(* CODESYS project MPS2017.project

Project tree, tasks and I/O mapping:
  Device : CECC-LK, Festo AG & Co. KG, order no. 574418, version 3.5.7.27
    application Application
      task Task (cyclic, interval 100 ms, priority 20) calls POU
      program POU [ST]
      global variables GVL
    Onboard : CECC 14I/8O, Festo AG & Co. KG, version 3.4.5.5
        unmapped channels: Onboard Input, Onboard Output
      Digital Inputs
          unmapped channels: Onboard Input
      Digital Outputs
          unmapped channels: Onboard Output
    Ethernet : Ethernet, 3S - Smart Software Solutions GmbH, version 3.5.7.0
        settings: IPAddress = [192,168,2,28]; SubnetMask = [255,255,255,0]; GatewayAddress = [0,0,0,0]; MACAddress = [16#00,16#00,16#00,16#00,16#00,16#00]; NetworkInterfaceName = 'eth0'; NetworkInterfaceName = "eth0"
      ModbusTCP_Slave_Device : ModbusTCP Slave Device, 3S - Smart Software Solutions GmbH, version 3.5.10.0
          settings: Unit-ID = 1; Data Model Options = 1
          input  Application.input1 AT %IW10 : ARRAY[0..11] OF WORD  // Inputs
          output Application.output1 AT %QW10 : ARRAY[0..11] OF WORD  // Outputs
    IO_Link_Master_4_Ports_ : IO-Link Master (4 Ports), Festo AG & Co. KG, order no. 
      , version 3.0.0.3
      BNI_IOL_310_000_K025 : BNI IOL-310-000-K025, BALLUFF, version V1.3
          settings:  = 0; ProcessDataID = V_PdT; ProcessDataInLength = 16; ProcessDataOutLength = 16; ProcessDataDescription.bitOffset = 8; ProcessDataDescription.bitLength = 1; ProcessDataDescription.userType = 0; ProcessDataDescription.ChannelType = 1; ProcessDataDescription.TotalLength = 16; ProcessDataDescription.bitOffset = 9; ProcessDataDescription.bitLength = 1; ProcessDataDescription.userType = 0; ProcessDataDescription.ChannelType = 1; ProcessDataDescription.TotalLength = 16; ProcessDataDescription.bitOffset = 10; ProcessDataDescription.bitLength = 1; ProcessDataDescription.userType = 0; ProcessDataDescription.ChannelType = 1; ProcessDataDescription.TotalLength = 16; ProcessDataDescription.bitOffset = 11; ProcessDataDescription.bitLength = 1; ProcessDataDescription.userType = 0; ProcessDataDescription.ChannelType = 1; ProcessDataDescription.TotalLength = 16; ProcessDataDescription.bitOffset = 12; ProcessDataDescription.bitLength = 1; ProcessDataDescription.userType = 0; ProcessDataDescription.ChannelType = 1; ProcessDataDescription.TotalLength = 16; ProcessDataDescription.bitOffset = 13; ProcessDataDescription.bitLength = 1; ProcessDataDescription.userType = 0; ProcessDataDescription.ChannelType = 1; ProcessDataDescription.TotalLength = 16; ProcessDataDescription.bitOffset = 14; ProcessDataDescription.bitLength = 1; ProcessDataDescription.userType = 0; ProcessDataDescription.ChannelType = 1; ProcessDataDescription.TotalLength = 16; ProcessDataDescription.bitOffset = 15;
            ProcessDataDescription.bitLength = 1; ProcessDataDescription.userType = 0; ProcessDataDescription.ChannelType = 1; ProcessDataDescription.TotalLength = 16; ProcessDataDescription.bitOffset = 0; ProcessDataDescription.bitLength = 1; ProcessDataDescription.userType = 0; ProcessDataDescription.ChannelType = 1; ProcessDataDescription.TotalLength = 16; ProcessDataDescription.bitOffset = 1; ProcessDataDescription.bitLength = 1; ProcessDataDescription.userType = 0; ProcessDataDescription.ChannelType = 1; ProcessDataDescription.TotalLength = 16; ProcessDataDescription.bitOffset = 2; ProcessDataDescription.bitLength = 1; ProcessDataDescription.userType = 0; ProcessDataDescription.ChannelType = 1; ProcessDataDescription.TotalLength = 16; ProcessDataDescription.bitOffset = 3; ProcessDataDescription.bitLength = 1; ProcessDataDescription.userType = 0; ProcessDataDescription.ChannelType = 1; ProcessDataDescription.TotalLength = 16; ProcessDataDescription.bitOffset = 4; ProcessDataDescription.bitLength = 1; ProcessDataDescription.userType = 0; ProcessDataDescription.ChannelType = 1; ProcessDataDescription.TotalLength = 16; ProcessDataDescription.bitOffset = 5; ProcessDataDescription.bitLength = 1; ProcessDataDescription.userType = 0; ProcessDataDescription.ChannelType = 1; ProcessDataDescription.TotalLength = 16; ProcessDataDescription.bitOffset = 6; ProcessDataDescription.bitLength = 1; ProcessDataDescription.userType = 0; ProcessDataDescription.ChannelType = 1; ProcessDataDescription.TotalLength = 16; ProcessDataDescription.bitOffset = 7;
            ProcessDataDescription.bitLength = 1; ProcessDataDescription.userType = 0; ProcessDataDescription.ChannelType = 1; ProcessDataDescription.TotalLength = 16; ProcessDataDescription.bitOffset = 8; ProcessDataDescription.bitLength = 1; ProcessDataDescription.userType = 0; ProcessDataDescription.ChannelType = 2; ProcessDataDescription.TotalLength = 16; ProcessDataDescription.bitOffset = 9; ProcessDataDescription.bitLength = 1; ProcessDataDescription.userType = 0; ProcessDataDescription.ChannelType = 2; ProcessDataDescription.TotalLength = 16; ProcessDataDescription.bitOffset = 10; ProcessDataDescription.bitLength = 1; ProcessDataDescription.userType = 0; ProcessDataDescription.ChannelType = 2; ProcessDataDescription.TotalLength = 16; ProcessDataDescription.bitOffset = 11; ProcessDataDescription.bitLength = 1; ProcessDataDescription.userType = 0; ProcessDataDescription.ChannelType = 2; ProcessDataDescription.TotalLength = 16; ProcessDataDescription.bitOffset = 12; ProcessDataDescription.bitLength = 1; ProcessDataDescription.userType = 0; ProcessDataDescription.ChannelType = 2; ProcessDataDescription.TotalLength = 16; ProcessDataDescription.bitOffset = 13; ProcessDataDescription.bitLength = 1; ProcessDataDescription.userType = 0; ProcessDataDescription.ChannelType = 2; ProcessDataDescription.TotalLength = 16; ProcessDataDescription.bitOffset = 14; ProcessDataDescription.bitLength = 1; ProcessDataDescription.userType = 0; ProcessDataDescription.ChannelType = 2; ProcessDataDescription.TotalLength = 16; ProcessDataDescription.bitOffset = 15;
            ProcessDataDescription.bitLength = 1; ProcessDataDescription.userType = 0; ProcessDataDescription.ChannelType = 2; ProcessDataDescription.TotalLength = 16; ProcessDataDescription.bitOffset = 0; ProcessDataDescription.bitLength = 1; ProcessDataDescription.userType = 0; ProcessDataDescription.ChannelType = 2; ProcessDataDescription.TotalLength = 16; ProcessDataDescription.bitOffset = 1; ProcessDataDescription.bitLength = 1; ProcessDataDescription.userType = 0; ProcessDataDescription.ChannelType = 2; ProcessDataDescription.TotalLength = 16; ProcessDataDescription.bitOffset = 2; ProcessDataDescription.bitLength = 1; ProcessDataDescription.userType = 0; ProcessDataDescription.ChannelType = 2; ProcessDataDescription.TotalLength = 16; ProcessDataDescription.bitOffset = 3; ProcessDataDescription.bitLength = 1; ProcessDataDescription.userType = 0; ProcessDataDescription.ChannelType = 2; ProcessDataDescription.TotalLength = 16; ProcessDataDescription.bitOffset = 4; ProcessDataDescription.bitLength = 1; ProcessDataDescription.userType = 0; ProcessDataDescription.ChannelType = 2; ProcessDataDescription.TotalLength = 16; ProcessDataDescription.bitOffset = 5; ProcessDataDescription.bitLength = 1; ProcessDataDescription.userType = 0; ProcessDataDescription.ChannelType = 2; ProcessDataDescription.TotalLength = 16; ProcessDataDescription.bitOffset = 6; ProcessDataDescription.bitLength = 1; ProcessDataDescription.userType = 0; ProcessDataDescription.ChannelType = 2; ProcessDataDescription.TotalLength = 16; ProcessDataDescription.bitOffset = 7;
            ProcessDataDescription.bitLength = 1; ProcessDataDescription.userType = 0; ProcessDataDescription.ChannelType = 2; ProcessDataDescription.TotalLength = 16
          unmapped channels: Switchstate Pin 1 (Bit0.0), Switchstate Pin 2 (Bit0.1), Switchstate Pin 3 (Bit0.2), Switchstate Pin 4 (Bit0.3), Switchstate Pin 5 (Bit0.4), Switchstate Pin 6 (Bit0.5), Switchstate Pin 7 (Bit0.6), Switchstate Pin 8 (Bit0.7), Switchstate Pin 9 (Bit1.0), Switchstate Pin 10 (Bit1.1), Switchstate Pin 11 (Bit1.2), Switchstate Pin 12 (Bit1.3), Switchstate Pin 13 (Bit1.4), Switchstate Pin 14 (Bit1.5), Switchstate Pin 15 (Bit1.6), Switchstate Pin 16 (Bit1.7), Switchstate Pin 1 (Bit0.0), Switchstate Pin 2 (Bit0.1), Switchstate Pin 3 (Bit0.2), Switchstate Pin 4 (Bit0.3), Switchstate Pin 5 (Bit0.4), Switchstate Pin 6 (Bit0.5), Switchstate Pin 7 (Bit0.6), Switchstate Pin 8 (Bit0.7), Switchstate Pin 9 (Bit1.0), Switchstate Pin 10 (Bit1.1), Switchstate Pin 11 (Bit1.2), Switchstate Pin 12 (Bit1.3), Switchstate Pin 13 (Bit1.4), Switchstate Pin 14 (Bit1.5), Switchstate Pin 15 (Bit1.6), Switchstate Pin 16 (Bit1.7)
      <Empty>
      <Empty>
      <Empty>
*)

// Device/Application/GVL
(* 
	Author: Alain Rohr (hftm.ch) / (Original by David Masternak(Festo)) 
	Date: 28.01.2017
*)

VAR_GLOBAL
	(** Variable for base station **)
	
	(* Input variables *)
	bs_partAtIn         AT %IX0.4 : BOOL;  (* Is part available on the left/in side *)
	bs_partAtOut        AT %IX0.6 : BOOL;  (* Is part available on the right/out side *)
	bs_base1Av          AT %IX2.2 : BOOL;  (* Are workpieces at output1 available *)
	bs_base2Av          AT %IX2.6 : BOOL;  (* Are workpieces at output2 available *)
	bs_base3Av          AT %IX0.2 : BOOL;  (* Are workpieces at output3 available *)
	bs_b1Retracted      AT %IX2.0 : BOOL;  (* Is Base1 Slide retracted *)
	bs_b1Extracted      AT %IX2.1 : BOOL;  (* Is Base1 Slide retracted *)
	
	bs_b2Retracted      AT %IX2.4 : BOOL;  (* Is Base2 Slide retracted *)
	bs_b2Extracted      AT %IX2.5 : BOOL;  (* Is Base2 Slide retracted *)
	
	bs_b3Retracted      AT %IX0.0 : BOOL;  (* Is Base3 Slide retracted *)
	bs_b3Extracted      AT %IX0.1 : BOOL;  (* Is Base3 Slide retracted *)
	
	(* Output variables *)
	bs_output1          AT %QX2.0 : BOOL;  (* Get workpiece at output1 *)
	bs_output2          AT %QX2.4 : BOOL;  (* Get workpiece at output2 *)
	bs_output3          AT %QX0.0 : BOOL;  (* Get workpiece at output3 *)
	
	bs_motorToOut       AT %QX0.4 : BOOL;  (* Run bandmotor to the left side *)
	bs_motorToIn        AT %QX0.5 : BOOL;  (* Run bandmotor to the right side *)
	bs_lightRed         AT %QX2.5 : BOOL;  (* Red light *)
	bs_lightYellow      AT %QX2.6 : BOOL;  (* Yellow light *)
	bs_lightGreen       AT %QX2.7 : BOOL;  (* Green light *)

	(** Variable for Ring-Station (pick and place 2) **)

	(* Input variables *)
	rs_partAtIn         AT %IX2.0 : BOOL;  (* Part available *)
	rs_partAtSep        AT %IX2.1 : BOOL;  (* Part at seperator *)
	rs_partAtOut        AT %IX2.2 : BOOL;  (* Part at delivery *)
	rs_partAtSlide      AT %IX2.3 : BOOL;  (* Part at slide *)

	rs_slide1Retracted  AT %IX2.4 : BOOL;  (* is slide1 extracted *)
	rs_slide1Extracted  AT %IX2.5 : BOOL;  (* is slide2 extracted *)
    rs_vacuum1IsOn      AT %IX2.6 : BOOL;  (* Eco trigger for slide 1 *)    

    rs_slide2Retracted  AT %IX0.0 : BOOL;  (* is slide2 retracted *)	
    rs_slide2Extracted  AT %IX0.1 : BOOL;  (* is slide2 extracted *)	
	rs_vacuum2IsOn      AT %IX0.2 : BOOL;  (* Eco trigger for slide 2 *)
	
	(* Output variables *)
	rs_motorToOut       AT %QX2.0 : BOOL;  (* Turn on bandmotor to Out *)
	rs_seperator        AT %QX2.2 : BOOL;  (* Turn on seperator *)
	
	rs_slide1Retract    AT %QX2.4 : BOOL;  (* Retract slide 1 *)
	rs_slide1Extract    AT %QX2.5 : BOOL;  (* Extend slide 1 *)
	rs_slide1Down       AT %QX2.6 : BOOL;  (* Up/Down slide 1 *)
	rs_vacuum1On        AT %QX0.6 : BOOL;  (* Vacuum on at slide 1 *)
	rs_vacuum1Off       AT %QX0.7 : BOOL;  (* Vacuum off at slide 1 *)
	
	rs_slide2Retract    AT %QX0.0 : BOOL;  (* Retract slide 2 *)
	rs_slide2Extract    AT %QX0.1 : BOOL;  (* Extend slide 2 *)
	rs_slide2Down       AT %QX0.2 : BOOL;  (* Up/Down slide 2 *)
	rs_vacuum2On        AT %QX0.4 : BOOL;  (* Vacuum on at slide 2 *)
	rs_vacuum2Off       AT %QX0.5 : BOOL;  (* Vacuum off at slide 2 *)
	
	rs_lightRed         AT %QX0.3 : BOOL;  (* Red light *)
	rs_lightYellow      AT %QX2.6 : BOOL;  (* Yellow light *)
	rs_lightGreen       AT %QX2.7 : BOOL;  (* Green light *)
	

	(** Variable for Cap Station (pick and place 1) **)
	(* Input variables *)
    cs_vacuumIsOn       AT %IX0.0 : BOOL;  (* Is Eco trigger active *)	
    cs_partAtIn         AT %IX2.0 : BOOL;  (* Is part available *)
	cs_partAtSep        AT %IX2.1 : BOOL;  (* Is part at seperator *)
	cs_partAtOut	    AT %IX2.2 : BOOL;  (* Is part on delivery position *)
	cs_slideRetracted   AT %IX2.4 : BOOL;
	cs_slideExtracted   AT %IX2.5 : BOOL;
	cs_slideIsUp	    AT %IX2.6 : BOOL;  (*Cylinder Z-Achse*)
	
	(* Output variables *)
	cs_vacuumOn	        AT %QX0.0 : BOOL;  (* Turn on vacuum *)
	cs_vacuumOff        AT %QX0.1 : BOOL;  (* Turn off vacuum *)
	cs_lightRed         AT %QX0.5 : BOOL;  (* Red light *)
	cs_lightYellow      AT %QX0.6 : BOOL;  (* Yellow light *)
	cs_lightGreen       AT %QX0.7 : BOOL;  (* Green light *)
	
	cs_motorToOut       AT %QX2.0 : BOOL;  (* Bandmotor *)
	cs_motorToIn        AT %QX2.1 : BOOL;  (* Bandmotor in other direction *)
	cs_seperator        AT %QX2.2 : BOOL;  (* Seperator *)
	cs_slideRetract     AT %QX2.4 : BOOL;  (* Retract slide *)
	cs_slideExtract     AT %QX2.5 : BOOL;  (* Extract slide *)
	cs_slideDown        AT %QX2.6 : BOOL;  (* Set slide down *)
	
	(** Variable for delivery station **)
	(*  Input variables *)
	ds_partAtIn         AT %IX0.0 : BOOL;  (* Part available *)
	ds_partAtInInd		AT %IX0.1 : BOOL;  (* inductive sensor*)
	ds_partAtIn2		AT %IX0.2 : BOOL;  (* Part sensor 2 *)
	ds_partAtOut        AT %IX0.3 : BOOL;  (* Part delivered *)
	ds_sep1Retracted	AT %IX0.4 : BOOL;
	ds_sep1Extracted	AT %IX0.5 : BOOL;
	ds_sep2Retracted	AT %IX0.6 : BOOL;
	ds_sep2Extracted	AT %IX0.7 : BOOL;	
	
	(* Output variables *)
	ds_motorToOut       AT %QX0.0 : BOOL;  (* Turn on bandmotor *)
	ds_sep1             AT %QX0.1 : BOOL;  (* Seperator line 1 *)
	ds_sep2             AT %QX0.2 : BOOL;  (* Seperator line 2 *)
	ds_lock             AT %QX0.3 : BOOL;  (* Lock at the beginning of band *)
	ds_lightRed         AT %QX2.5 : BOOL;  (* Red light *)
	ds_lightYellow      AT %QX2.6 : BOOL;  (* Yellow light *)
	ds_lightGreen       AT %QX2.7 : BOOL;  (* Green light *)
	
	

	(* Variable for all mps types *)
	mpsType : INT := 1; (* What kind of machine *)
	SFCInit : BOOL;
	SFCCurrentStep : STRING;
	
	(** MODBUS stuff **)
	input1  : ARRAY[0..11] OF WORD; (* Modbus input register *)
	output1 : ARRAY[0..11] OF WORD; (* Modbus output register *)
	
	(*CDP*)
	flanke:BOOL; (*Flankenspiel für Processing*)
	sensorSpiel:BOOL; (*FlankenSpiel für Werkstückerkennung*)
	noRefBox:BOOL:=TRUE;
	uiStep: UINT; (*Variable für Schrittweise durchführung von Maschine 0*)
	
	(*other Global Variables*)
	rs_slideCounter : INT := 0;
	bs_lastInput : WORD := 0;
    bs_delayTime : TIME := T#0.0S; (* Delaytime for different workpiece colors *)
    bs_delSiteToOut             : INT := 0; (* On what side we want to deliver (out if 1 / in if 0) *)
	
	(* Just for debugging *)
	rs_t17 AT %IX0.0 : BOOL;
	rs_t18 AT %IX0.1 : BOOL;
	rs_t19 AT %IX0.2 : BOOL;
	rs_t20 AT %IX0.3 : BOOL;
	rs_t21 AT %IX0.4 : BOOL;
	rs_t22 AT %IX0.5 : BOOL;
	rs_t23 AT %IX0.6 : BOOL;
	rs_t24 AT %IX0.7 : BOOL;
	rs_t25 AT %IX2.0 : BOOL;
	rs_t26 AT %IX2.1 : BOOL;
	rs_t27 AT %IX2.2 : BOOL;
	rs_t28 AT %IX2.3 : BOOL;
	rs_t29 AT %IX2.4 : BOOL;
	rs_t30 AT %IX2.5 : BOOL;
	rs_t31 AT %IX2.6 : BOOL;
	rs_t32 AT %IX2.7 : BOOL;
	rs_t33 AT %QX3.0 : BOOL;
	rs_t34 AT %QX3.1 : BOOL;
	rs_t35 AT %QX3.2 : BOOL;
	rs_t36 AT %QX3.3 : BOOL;
	rs_t37 AT %QX3.4 : BOOL;
	rs_t38 AT %QX3.5 : BOOL;
	rs_t39 AT %QX3.6 : BOOL;
	rs_t40 AT %QX3.7 : BOOL;
	rs_slide : INT;
END_VAR

// Device/Application/POU
PROGRAM POU
VAR CONSTANT
	BS: WORD := 1;
	RS: WORD := 2;
	CS: WORD := 3;
	DS: WORD := 4;
	SS: WORD := 5;
END_VAR

VAR
	x1: BOOL;
END_VAR

GVL.input1[10]:=DS;

CASE GVL.input1[10] OF
	BS:
	  GVL.bs_motorToOut:=GVL.input1[0].0;
	  GVL.bs_motorToIn:=GVL.input1[0].1;
	  GVL.bs_lightRed:=GVL.input1[0].5;
	  GVL.bs_lightYellow:=GVL.input1[0].6;
	  GVL.bs_lightGreen:=GVL.input1[0].7;
	  GVL.bs_output1:=GVL.input1[0].8;
	  GVL.bs_output2:=GVL.input1[0].9;
	  GVL.bs_output3:=GVL.input1[0].10;
	  
	  GVL.output1[0].0:=GVL.bs_partAtIn;
	  GVL.output1[0].2:=GVL.bs_partAtOut;
	  GVL.output1[0].4:=GVL.bs_b1Retracted;
	  GVL.output1[0].5:=GVL.bs_b1Extracted;
	  GVL.output1[0].6:=GVL.bs_b2Retracted;
	  GVL.output1[0].7:=GVL.bs_b2Extracted;
	  GVL.output1[0].8:=GVL.bs_b3Retracted;
	  GVL.output1[0].9:=GVL.bs_b3Extracted;
	  GVL.output1[0].10:=GVL.bs_base1Av;
	  GVL.output1[0].11:=GVL.bs_base2Av;
	  GVL.output1[0].12:=GVL.bs_base3Av;
	  
	RS:
	  GVL.rs_motorToOut:=GVL.input1[0].0;
	  GVL.rs_seperator:=GVL.input1[0].2;
	  GVL.rs_lightRed:=GVL.input1[0].5;
	  GVL.rs_lightYellow:=GVL.input1[0].6;
	  GVL.rs_lightGreen:=GVL.input1[0].7;
	  GVL.rs_slide1Retract:=GVL.input1[0].8;
	  GVL.rs_slide1Extract:=GVL.input1[0].9;
	  GVL.rs_slide1Down:=GVL.input1[0].10;
	  GVL.rs_vacuum1On:=GVL.input1[0].11;
	  GVL.rs_vacuum1Off:=GVL.input1[0].12;
	  GVL.rs_slide2Retract:=GVL.input1[1].0;
	  GVL.rs_slide2Extract:=GVL.input1[1].1;
	  GVL.rs_slide2Down:=GVL.input1[1].2;
	  GVL.rs_vacuum2On:=GVL.input1[1].3;
	  GVL.rs_vacuum2Off:=GVL.input1[1].4;
	  
	  GVL.output1[0].0:=GVL.rs_partAtIn;
	  GVL.output1[0].1:=GVL.rs_partAtSep;
	  GVL.output1[0].2:=GVL.rs_partAtOut;
	  GVL.output1[0].3:=GVL.rs_partAtSlide;
	  GVL.output1[0].4:=GVL.rs_slide1Retracted;
	  GVL.output1[0].5:=GVL.rs_slide1Extracted;
	  GVL.output1[0].6:=GVL.rs_slide2Retracted;
	  GVL.output1[0].7:=GVL.rs_slide2Extracted;
	  GVL.output1[0].10:=GVL.rs_vacuum1IsOn;
	  GVL.output1[0].11:=GVL.rs_vacuum2IsOn;
	  
	CS:
	  GVL.cs_motorToOut:=GVL.input1[0].0;
	  GVL.cs_motorToIn:=GVL.input1[0].1;
	  GVL.cs_seperator:=GVL.input1[0].2;
	  GVL.cs_lightRed:=GVL.input1[0].5;
	  GVL.cs_lightYellow:=GVL.input1[0].6;
	  GVL.cs_lightGreen:=GVL.input1[0].7;
	  GVL.cs_slideRetract:=GVL.input1[0].8;
	  GVL.cs_slideExtract:=GVL.input1[0].9;
	  GVL.cs_slideDown:=GVL.input1[0].10;
	  GVL.cs_vacuumOn:=GVL.input1[0].11;
	  GVL.cs_vacuumOff:=GVL.input1[0].12;
	  
	  GVL.output1[0].0:=GVL.cs_partAtIn;
	  GVL.output1[0].1:=GVL.cs_partAtSep;
	  GVL.output1[0].2:=GVL.cs_partAtOut;
	  GVL.output1[0].3:=GVL.cs_slideIsUp;
	  GVL.output1[0].4:=GVL.cs_slideRetracted;
	  GVL.output1[0].5:=GVL.cs_slideExtracted;
	  GVL.output1[0].10:=GVL.cs_vacuumIsOn;
	  
	DS:
	  GVL.ds_motorToOut:=GVL.input1[0].0;
	  GVL.ds_sep1:=GVL.input1[0].2;
	  GVL.ds_sep2:=GVL.input1[0].3;
	  GVL.ds_lightRed:=GVL.input1[0].5;
	  GVL.ds_lightYellow:=GVL.input1[0].6;
	  GVL.ds_lightGreen:=GVL.input1[0].7;	
	  
	  GVL.output1[0].0:=GVL.ds_partAtIn;
	  GVL.output1[0].2:=GVL.ds_partAtOut;
	  GVL.output1[0].4:=GVL.ds_sep1Retracted;
	  GVL.output1[0].5:=GVL.ds_sep1Extracted;
	  GVL.output1[0].6:=GVL.ds_sep2Retracted;
	  GVL.output1[0].7:=GVL.ds_sep2Extracted;
	SS:	  
	  //not yet implemented
END_CASE

END_PROGRAM
